FUNCTION_BLOCK FB_TDS3000 EXTENDS FB_ModbusSlave
VAR
	arrConditionData	:	ARRAY [0..63] OF WORD;
	arrUp_LoLimit		:	ARRAY [0..63] OF WORD;
	arrUpUp_UpLimit		:	ARRAY [0..63] OF WORD;
END_VAR

PROPERTY ConditionData : ARRAY [0..63] OF WORD
GET
ConditionData := arrConditionData;
END_GET
END_PROPERTY

METHOD Convert : BOOL
VAR_INPUT
	iRegionNo	:	INT;
	pReadData	:	POINTER TO BYTE;
END_VAR
VAR
	pTempData	: 	POINTER TO BYTE;
	iTempData	: 	BYTE;
	iLoop		: 	INT;
	bHiByte		:	BOOL := TRUE;
END_VAR
CASE iRegionNo OF
	0: 
		FOR iLoop := 0 TO SIZEOF(arrAddress[0][1])*2 DO
			pTempData := (pReadData + iLoop);
			iTempData := pTempData^;
			
			IF bHiByte THEN
				arrConditionData[iLoop/2] := SHL(BYTE_TO_WORD(iTempData), 8);
			ELSE 
				arrConditionData[iLoop/2] := arrConditionData[iLoop/2] + BYTE_TO_WORD(iTempData);
				IF bSwap THEN
					arrConditionData[iLoop/2] := ROL(arrConditionData[iLoop/2], 8);
				END_IF
			END_IF
			bHiByte := NOT bHiByte;
		END_FOR
		
	1:
		FOR iLoop := 17 TO (SIZEOF(arrAddress[1][1])*2 + 17) DO
			pTempData := (pReadData + iLoop);
			iTempData := pTempData^;
			
			IF bHiByte THEN
				arrConditionData[iLoop/2] := SHL(BYTE_TO_WORD(iTempData), 8);
			ELSE 
				arrConditionData[iLoop/2] := arrConditionData[iLoop/2] + BYTE_TO_WORD(iTempData);
				IF bSwap THEN
					arrConditionData[iLoop/2] := ROL(arrConditionData[iLoop/2], 8);
				END_IF
			END_IF
			bHiByte := NOT bHiByte;
		END_FOR
		
	2: 
		FOR iLoop := 0 TO SIZEOF(arrAddress[2][1])*2 DO
			pTempData := (pReadData + iLoop);
			iTempData := pTempData^;
			
			IF bHiByte THEN
				arrUp_LoLimit[iLoop/2] := SHL(BYTE_TO_WORD(iTempData), 8);
			ELSE 
				arrUp_LoLimit[iLoop/2] := arrUp_LoLimit[iLoop/2] + BYTE_TO_WORD(iTempData);
				IF bSwap THEN
					arrUp_LoLimit[iLoop/2] := ROL(arrUp_LoLimit[iLoop/2], 8);
				END_IF
			END_IF
			bHiByte := NOT bHiByte;
		END_FOR
		
	3: 
		FOR iLoop := 17 TO SIZEOF(arrAddress[3][1])*2 + 17 DO
			pTempData := (pReadData + iLoop);
			iTempData := pTempData^;
			
			IF bHiByte THEN
				arrUp_LoLimit[iLoop/2] := SHL(BYTE_TO_WORD(iTempData), 8);
			ELSE 
				arrUp_LoLimit[iLoop/2] := arrUp_LoLimit[iLoop/2] + BYTE_TO_WORD(iTempData);
				IF bSwap THEN
					arrUp_LoLimit[iLoop/2] := ROL(arrUp_LoLimit[iLoop/2], 8);
				END_IF
			END_IF
			bHiByte := NOT bHiByte;
		END_FOR

	4: 
		FOR iLoop := 0 TO SIZEOF(arrAddress[4][1])*2 DO
			pTempData := (pReadData + iLoop);
			iTempData := pTempData^;
			
			IF bHiByte THEN
				arrUpUp_UpLimit[iLoop/2] := SHL(BYTE_TO_WORD(iTempData), 8);
			ELSE 
				arrUpUp_UpLimit[iLoop/2] := arrUpUp_UpLimit[iLoop/2] + BYTE_TO_WORD(iTempData);
				IF bSwap THEN
					arrUpUp_UpLimit[iLoop/2] := ROL(arrUpUp_UpLimit[iLoop/2], 8);
				END_IF
			END_IF
			bHiByte := NOT bHiByte;
		END_FOR

	5: 
		FOR iLoop := 17 TO SIZEOF(arrAddress[5][1])*2 + 17 DO
			pTempData := (pReadData + iLoop);
			iTempData := pTempData^;
			
			IF bHiByte THEN
				arrUpUp_UpLimit[iLoop/2] := SHL(BYTE_TO_WORD(iTempData), 8);
			ELSE 
				arrUpUp_UpLimit[iLoop/2] := arrUpUp_UpLimit[iLoop/2] + BYTE_TO_WORD(iTempData);
				IF bSwap THEN
					arrUpUp_UpLimit[iLoop/2] := ROL(arrUpUp_UpLimit[iLoop/2], 8);
				END_IF
			END_IF
			bHiByte := NOT bHiByte;
		END_FOR

END_CASE
END_METHOD

METHOD FirstCycle : BOOL
VAR_INPUT
END_VAR
arrAddress[0][0] := 16#0000;
arrAddress[0][1] := 17;
arrAddress[1][0] := 16#0017;
arrAddress[1][1] := 15;

arrAddress[2][0] := 16#0100;
arrAddress[2][1] := 17;
arrAddress[3][0] := 16#0117;
arrAddress[3][1] := 15;

arrAddress[4][0] := 16#0200;
arrAddress[4][1] := 17;
arrAddress[5][0] := 16#0217;
arrAddress[5][1] := 15;

iNumAddRegion := 6;

bSwap := TRUE;
END_METHOD

PROPERTY Up_LoLimit : ARRAY [0..63] OF WORD
GET
Up_LoLimit := arrUp_LoLimit;
END_GET
END_PROPERTY

PROPERTY UpUp_UpLimit : ARRAY [0..63] OF WORD
GET
UpUp_UpLimit := arrUpUp_UpLimit;
END_GET
END_PROPERTY

END_FUNCTION_BLOCK

(* stored: Version 1.1.0.1, ProductVersion 3.1.4024.12
   POU FB_TDS3000: Id {e8fb70df-be29-4460-957f-9586549f42be}, SpecialFunc None
   Property ConditionData: Id {f85b153e-777c-46bf-afd8-d7a098fe9e2d}
   Get Get: Id {a26145bd-6d63-412a-ae13-c34a1165bf75}
   Method Convert: Id {b48e17b2-54ba-4775-8ece-9ac9c943983a}
   Method FirstCycle: Id {70eeedf9-dc8a-4bd4-9ac7-1fc925a31989}
   Property Up_LoLimit: Id {d5b8ab1e-d642-46de-8c6b-98e1a26d2cb6}
   Get Get: Id {e20bdbc2-bf8e-4486-913d-26f0a21b8c5f}
   Property UpUp_UpLimit: Id {c107981f-2291-4349-8d24-74209dc61e7b}
   Get Get: Id {6abb6c8a-f004-493f-b539-3cad41bef48c} *)
